Staubli VAL3: RobotStatus.pjx

--- RobotStatus.pjx ---
Parameters version=s7.7.2 stackSize=5000 millimeterUnit=true
Program file=start.pgx
Program file=stop.pgx
Data file=RobotStatus.dtx

--- RobotStatus.dtx ---
public num nDrivesPowered
public num nEStopped
public num nErrorCode
public num nInError
public num nInMotion
public num nMode
public num nMotionPossible
